(* IEC 61131-3 sources: AXOpen/src/components.rexroth.drives/ctrl/src/AxoCtrlxDriveXsc/v_6_x_x/TypesStructuresAndEnums, 13 files *)

(* ---- AxoCtrlxDriveXsc_Component_Status.st ---- *)
NAMESPACE AXOpen.Components.Rexroth.Drives.v_6_x_x
    {S7.extern=ReadWrite}
    {#ix-attr:[Container(Layout.Stack)]}
    CLASS PUBLIC AxoCtrlxDriveXsc_Component_Status EXTENDS AXOpen.Components.Drives.AxoDrive_Status
        VAR PUBLIC

        END_VAR
    END_CLASS
END_NAMESPACE

(* ---- AxoCtrlxDriveXsc_Config.st ---- *)
NAMESPACE AXOpen.Components.Rexroth.Drives.v_6_x_x
    {S7.extern=ReadWrite}
    {#ix-attr:[Container(Layout.Stack)]}
    CLASS PUBLIC AxoCtrlxDriveXsc_Config
        VAR PUBLIC
            {#ix-set:AttributeName = "<#Info time#>"}
            InfoTime : LTIME := LT#5S;
            {#ix-set:AttributeName = "<#Error time#>"}
            ErrorTime : LTIME := LT#10S;
            {#ix-set:AttributeName = "<#Task timeout#>"}
            TaskTimeout : LTIME := LT#50S;
        END_VAR
    END_CLASS
END_NAMESPACE

(* ---- AxoCtrlxDriveXsc_Control.st ---- *)
NAMESPACE AXOpen.Components.Rexroth.Drives.v_6_x_x
    {S7.extern=ReadWrite}
    {#ix-attr:[Container(Layout.Tabs)]}
    CLASS PUBLIC AxoCtrlxDriveXsc_Control
        VAR PUBLIC
            {#ix-set:AttributeName = "<#DriveControlWord_S_0_0134_0_0#>"}
            DriveControlWord_S_0_0134_0_0 : AxoCtrlxDriveXscDriveControlWord_S_0_0134_0_0;
            {#ix-set:AttributeName = "<#SignalControlWord_S_0_0145_0_0#>"}
            SignalControlWord_S_0_0145_0_0 :    AxoCtrlxDriveXscSignalControlWord_S_0_0145_0_0;
            {#ix-set:AttributeName = "<#CommandPosition_S_0_0282_0_0#>"}
            CommandPosition_S_0_0282_0_0 : DINT;
            {#ix-set:AttributeName = "<#CommandVelocity_S_0_0259_0_0#>"}
            CommandVelocity_S_0_0259_0_0 : DINT;
            {#ix-set:AttributeName = "<#CommandAcceleration_S_0_0260_0_0#>"}
            CommandAcceleration_S_0_0260_0_0 : DINT;
            {#ix-set:AttributeName = "<#CommandDecceleration_S_0_0359_0_0#>"}
            CommandDecceleration_S_0_0359_0_0 : DINT;
            {#ix-set:AttributeName = "<#SupplyUnitControlWord_S_0_1720_0_1#>"}
            SupplyUnitControlWord_S_0_1720_0_1  : AxoCtrlxDriveXscSupplyUnitControlWord_S_0_1720_0_1;
            {#ix-set:AttributeName = "<#BipolarTorqueLimitation_S_0_0092_0_0#>"}
            BipolarTorqueLimitation_S_0_0092_0_0: INT;
            {#ix-set:AttributeName = "<#CommandTorque_S_0_0080_0_0#>"}
            CommandTorque_S_0_0080_0_0 : INT;
            {#ix-set:AttributeName = "<#CommandJerk_S_0_0193_0_0#>"}
            CommandJerk_S_0_0193_0_0 : DINT;
        END_VAR
    END_CLASS
END_NAMESPACE

(* ---- AxoCtrlxDriveXsc_Status.st ---- *)
NAMESPACE AXOpen.Components.Rexroth.Drives.v_6_x_x
    {S7.extern=ReadWrite}
    {#ix-attr:[Container(Layout.Tabs)]}
    CLASS PUBLIC AxoCtrlxDriveXsc_Status
        VAR PUBLIC
            {#ix-set:AttributeName = "<#DriveStatusWord_S_0_0135_0_0#>"}
            DriveStatusWord_S_0_0135_0_0 : AxoCtrlxDriveXscDriveStatusWord_S_0_0135_0_0;
            {#ix-set:AttributeName = "<#SignalStatusWord_S_0_0144_0_0#>"}
            SignalStatusWord_S_0_0144_0_0 : AxoCtrlxDriveXscSignalStatusWord_S_0_0144_0_0;
            {#ix-set:AttributeName = "<#ActualPosition_S_0_0386_0_0#>"}
            ActualPosition_S_0_0386_0_0 : DINT;
            {#ix-set:AttributeName = "<#ActualVelocity_S_0_0535_0_0#>"}
            ActualVelocity_S_0_0535_0_0 : DINT;
            {#ix-set:AttributeName = "<#DiagnosticMessage_S_0_0390_0_0#>"}
            DiagnosticMessage_S_0_0390_0_0 : DWORD;
            {#ix-set:AttributeName = "<#SupplyUnitStatusWord_S_0_1720_0_2#>"}
            SupplyUnitStatusWord_S_0_1720_0_2 : AxoCtrlxDriveXscSupplyUnitStatusWord_S_0_1720_0_2;
            {#ix-set:AttributeName = "<#ActualTorque_S_0_0084_0_0#>"}
            ActualTorque_S_0_0084_0_0 : INT;
        END_VAR
    END_CLASS
END_NAMESPACE

(* ---- AxoCtrlxDriveXscAxisData.st ---- *)
NAMESPACE AXOpen.Components.Rexroth.Drives.v_6_x_x
    {S7.extern=ReadWrite}
    CLASS AxoCtrlxDriveXscAxisData
        VAR PUBLIC
            Cycle                       :   ULINT;
            OverrideVelocityFactor		:	LREAL := 1.0;	//LREAL value to be written
            OverrideAccelerationFactor	:	LREAL := 1.0;	//LREAL value to be written
            OverrideJerkFactor			:	LREAL := 1.0;	//LREAL value to be written
        END_VAR
    END_CLASS
END_NAMESPACE

(* ---- AxoCtrlxDriveXscAxisReference.st ---- *)
// USING AXOpen.Components.Drives;

NAMESPACE AXOpen.Components.Rexroth.Drives.v_6_x_x
    {S7.extern=ReadWrite}
    CLASS AxoCtrlxDriveXscAxisReference IMPLEMENTS AXOpen.Components.Abstractions.Drives.IAxoAxisReference
        VAR PUBLIC // HWin
            {#ix-attr:[Container(Layout.Stack)]}
            {#ix-attr:[ComponentDetails("HW inputs")]}
            {#ix-attr:[ReadOnly()]}
            Inputs  :   AxoCtrlxDriveXsc_Status;
        END_VAR
        VAR PUBLIC // HWout
            {#ix-attr:[Container(Layout.Stack)]}
            {#ix-attr:[ComponentDetails("HW outputs")]}
            // {#ix-attr:[ReadOnly()]}
            Outputs  :   AxoCtrlxDriveXsc_Control;
        END_VAR
        VAR PUBLIC // HWIDs
            {#ix-attr:[Container(Layout.Stack)]}
            {#ix-attr:[ComponentDetails("HWids")]}
            {#ix-attr:[ReadOnly()]}
            HWIDs  :   AxoCtrlxDriveXscHWIDs;
        END_VAR
        VAR PUBLIC // Data
            {#ix-attr:[Container(Layout.Stack)]}
            {#ix-attr:[ComponentDetails("Data")]}
            {#ix-attr:[ReadOnly()]}
            Data            :   AxoCtrlxDriveXscAxisData;
        END_VAR
        VAR PUBLIC
            Config          :   AXOpen.Components.Drives.AxoDrive_Config;
            Status          :   AXOpen.Components.Drives.AxoDrive_Status;
        END_VAR
    END_CLASS
END_NAMESPACE

(* ---- AxoCtrlxDriveXscDriveControlWord_S_0_0134_0_0.st ---- *)
NAMESPACE AXOpen.Components.Rexroth.Drives.v_6_x_x
    {S7.extern=ReadWrite}
    {#ix-attr:[Container(Layout.Wrap)]}
    {#ix-attr:[Group(GroupLayout.GroupBox)]}
    {#ix-set:AttributeName = "<#DriveControlWord#>"}
    CLASS AxoCtrlxDriveXscDriveControlWord_S_0_0134_0_0
        VAR PUBLIC
            {#ix-set:AttributeName = "<#_bit00_Reserve#>"}
            _bit00_Reserve 				:	BOOL;
            {#ix-set:AttributeName = "<#_bit01_Reserve#>"}
            _bit01_Reserve 				:	BOOL;
            {#ix-set:AttributeName = "<#_bit02_Reserve#>"}
            _bit02_Reserve 				:	BOOL;
            {#ix-set:AttributeName = "<#_bit03_Reserve#>"}
            _bit03_Reserve 				:	BOOL;
            {#ix-set:AttributeName = "<#_bit04_Reserve#>"}
            _bit04_Reserve 				:	BOOL;
            {#ix-set:AttributeName = "<#_bit05_Reserve#>"}
            _bit05_Reserve 				:	BOOL;
            {#ix-set:AttributeName = "<#_bit06_Reserve#>"}
            _bit06_Reserve 				:	BOOL;
            {#ix-set:AttributeName = "<#_bit07_Reserve#>"}
            _bit07_Reserve 				:	BOOL;

            {#ix-set:AttributeName = "<#Command operation mode Bit 0#>"}
            CommandOperationModeBit0 	:	BOOL;		//  Command operation mode bit 0                        |   000:  Primary operation mode
                                                        //                                                      |   001:  Secondary operation mode 1
            {#ix-set:AttributeName = "<#Command operation mode Bit 1#>"}
            CommandOperationModeBit1 	:	BOOL;		//  Command operation mode bit 1                        |   010:  Secondary operation mode 2
                                                        //                                                      |   011:  Secondary operation mode 3
                                                        //                                                      |   100:  Secondary operation mode 4
            {#ix-set:AttributeName = "<#Command operation mode Bit 2#>"}
            CommandOperationModeBit2 	:	BOOL;		//  Command operation mode bit 2                        |   101:  Secondary operation mode 5
                                                        //                                                      |   110:  Secondary operation mode 6
                                                        //                                                      |   111:  Secondary operation mode 7
            {#ix-set:AttributeName = "<#_bit11_Reserve#>"}
            _bit11_Reserve 				:	BOOL;
            {#ix-set:AttributeName = "<#_bit12_Reserve#>"}
            _bit12_Reserve 				:	BOOL;
            {#ix-set:AttributeName = "<#Drive Halt#>"}
            DriveHalt 				:	BOOL;		        //  1-0 change: Deceleration of drive while maintaining maximum acceleration (S‑0‑0138 - only possible if bits 14 and 15 = 1)
            {#ix-set:AttributeName = "<#Drive enable#>"}
            DriveEnable 				:	BOOL;		    //  Negative edge: Torque disable without delay (independent of bit 15 or 13)
            {#ix-set:AttributeName = "<#Drive On#>"}
            DriveOn 				:	BOOL;		        //  Negative edge: Best possible deceleration (only possible if bit 14 = 1)
        END_VAR
    END_CLASS
END_NAMESPACE

(* ---- AxoCtrlxDriveXscDriveStatusWord_S_0_0135_0_0.st ---- *)
NAMESPACE AXOpen.Components.Rexroth.Drives.v_6_x_x
    {S7.extern=ReadWrite}
    {#ix-attr:[Container(Layout.Wrap)]}
    {#ix-attr:[Group(GroupLayout.GroupBox)]}
    {#ix-set:AttributeName = "<#DriveStatusWord#>"}
    CLASS AxoCtrlxDriveXscDriveStatusWord_S_0_0135_0_0
        VAR PUBLIC
            {#ix-set:AttributeName = "<#_bit00_Reserve#>"}
            _bit00_Reserve 				:	BOOL;
            {#ix-set:AttributeName = "<#_bit01_Reserve#>"}
            _bit01_Reserve 				:	BOOL;
            {#ix-set:AttributeName = "<#_bit02_Reserve#>"}
            _bit02_Reserve 				:	BOOL;
            {#ix-set:AttributeName = "<#CommandProcessingStatus#>"}
            CommandProcessingStatus		:	BOOL;		//  0 - Drive ignores command value input           |   1 -Drive follows command value input
            {#ix-set:AttributeName = "<#InStandstill#>"}
            InStandstill 				:	BOOL;		//  Drive "Halt" status                             |   1- Act vel < standstill window
            {#ix-set:AttributeName = "<#InReference#>"}
            InReference 				:	BOOL;		//  Drive hommed
            {#ix-set:AttributeName = "<#_bit06_Reserve#>"}
            _bit06_Reserve 				:	BOOL;
            {#ix-set:AttributeName = "<#HardwareLock#>"}
            HardwareLock                :	BOOL;       //  Hardware lock (E-stop)
            {#ix-set:AttributeName = "<#ActualOperatingModeBit0#>"}
            ActualOperatingModeBit0 	:	BOOL;		//  Actual_operating mode bit 0                     |   000:  Primary operation mode
                                                        //                                                  |   001:  Secondary operation mode 1
            {#ix-set:AttributeName = "<#ActualOperatingModeBit1#>"}
            ActualOperatingModeBit1 	:	BOOL;		//  Actual_operating mode bit 1                     |   010:  Secondary operation mode 2
                                                        //                                                  |   011:  Secondary operation mode 3
                                                        //                                                  |   100:  Secondary operation mode 4
            {#ix-set:AttributeName = "<#ActualOperatingModeBit2#>"}
            ActualOperatingModeBit2 	:	BOOL;		//  Actual_operating mode bit 2                     |   101:  Secondary operation mode 5
                                                        //                                                  |   110:  Secondary operation mode 6
                                                        //                                                  |   111:  Secondary operation mode 7
            {#ix-set:AttributeName = "<#_bit11_Reserve#>"}
            _bit11_Reserve 				:	BOOL;
            {#ix-set:AttributeName = "<#WarningZKL2#>"}
            WarningZKL2 				:	BOOL;		//  Warning ZKL2
            {#ix-set:AttributeName = "<#DriveErrorZKL1#>"}
            DriveErrorZKL1 				:	BOOL;		//  Drive Error ZKL1
            {#ix-set:AttributeName = "<#ReadyForOperation Bit 0#>"}
            ReadyForOperationBit0       :	BOOL;		//  Ready to operate bit 0 lower significant bit    |   10: Control section and power section ready for op. (Ab)
                                                        //                                                  |   11: In operation, with torque (e.g. AF)
            {#ix-set:AttributeName = "<#ReadyForOperation Bit 1#>"}
            ReadyForOperationBit1       :	BOOL;		//  Ready to operate bit 1 higher significant bit   |   00: Not ready for power on (e.g., P2)
                                                        //                                                  |   01: Ready for power on (bb)
        END_VAR
    END_CLASS
END_NAMESPACE

(* ---- AxoCtrlxDriveXscHWIDs.st ---- *)
NAMESPACE AXOpen.Components.Rexroth.Drives.v_6_x_x
   {S7.extern=ReadWrite}
	CLASS AxoCtrlxDriveXscHWIDs
      VAR PUBLIC
         {#ix-set:AttributeName = "<#Hardware ID Device#>"}
         HW_Device            : UINT;
         {#ix-set:AttributeName = "<#Hardware ID 'Outputs' module#>"}
         HW_Outputs           : UINT;
         {#ix-set:AttributeName = "<#Hardware ID 'Inputs' module#>"}
         HW_Inputs            : UINT;
         {#ix-set:AttributeName = "<#Hardware ID 'S_0_0134_0_0__Servodrive_profile__Control_word' submodule#>"}
         HW_S_0_0134_0_0      : UINT;
         {#ix-set:AttributeName = "<#Hardware ID 'S_0_0145_0_0__Signal_control_word__Value' submodule#>"}
         HW_S_0_0145_0_0      : UINT;
         {#ix-set:AttributeName = "<#Hardware ID 'S_0_0282_0_0__Drive_controlled_positioning__Command_value' submodule#>"}
         HW_S_0_0282_0_0      : UINT;
         {#ix-set:AttributeName = "<#Hardware ID 'S_0_0259_0_0__Positioning_profile__Profile_velocity' submodule#>"}
         HW_S_0_0259_0_0      : UINT;
         {#ix-set:AttributeName = "<#Hardware ID 'S_0_0260_0_0__Positioning_profile__Acceleration' submodule#>"}
         HW_S_0_0260_0_0      : UINT;
         {#ix-set:AttributeName = "<#Hardware ID 'S_0_0359_0_0__Positioning_profile__Deceleration' submodule#>"}
         HW_S_0_0359_0_0      : UINT;
         {#ix-set:AttributeName = "<#Hardware ID 'S_0_1720_0_1__Power_supply_control__Control_word' submodule#>"}
         HW_S_0_1720_0_1      : UINT;
         {#ix-set:AttributeName = "<#Hardware ID 'S_0_0092_0_0__Torque_force_limitation__Limit_value_bipolar' submodule#>"}
         HW_S_0_0092_0_0      : UINT;
         {#ix-set:AttributeName = "<#Hardware ID 'S_0_0080_0_0__Torque_force_command_value' submodule#>"}
         HW_S_0_0080_0_0      : UINT;
         {#ix-set:AttributeName = "<#Hardware ID 'S_0_0193_0_0__Positioning_jerk' submodule#>"}
         HW_S_0_0193_0_0      : UINT;
         {#ix-set:AttributeName = "<#Hardware ID 'S_0_0135_0_0__Servodrive_profile__Status_word' submodule#>"}
         HW_S_0_0135_0_0      : UINT;
         {#ix-set:AttributeName = "<#Hardware ID 'S_0_0144_0_0__Signal_status_word__Value' submodule#>"}
         HW_S_0_0144_0_0      : UINT;
         {#ix-set:AttributeName = "<#Hardware ID 'S_0_0386_0_0__Position_controller__Position_actual_value' submodule#>"}
         HW_S_0_0386_0_0      : UINT;
         {#ix-set:AttributeName = "<#Hardware ID 'S_0_0535_0_0__Velocity_controller__Velocity_actual_value' submodule#>"}
         HW_S_0_0535_0_0      : UINT;
         {#ix-set:AttributeName = "<#Hardware ID 'S_0_0390_0_0__Diagnostic_message__Manufacturer_status_register' submodule#>"}
         HW_S_0_0390_0_0      : UINT;
         {#ix-set:AttributeName = "<#Hardware ID 'S_0_1720_0_2__Power_supply_control__Status_word' submodule#>"}
         HW_S_0_1720_0_2      : UINT;
         {#ix-set:AttributeName = "<#Hardware ID 'S_0_0084_0_0__Torque_force_feedback_value' submodule#>"}
         HW_S_0_0084_0_0      : UINT;
         {#ix-set:AttributeName = "<#Hardware ID 'P_0_0106_0_0__STO_function__Operating_status' submodule#>"}
         HW_P_0_0106_0_0      : UINT;
      END_VAR
   END_CLASS
END_NAMESPACE

(* ---- AxoCtrlxDriveXscSignalControlWord_S_0_0145_0_0.st ---- *)
NAMESPACE AXOpen.Components.Rexroth.Drives.v_6_x_x
    {S7.extern=ReadWrite}
    {#ix-attr:[Container(Layout.Wrap)]}
    {#ix-attr:[Group(GroupLayout.GroupBox)]}
    {#ix-set:AttributeName = "<#SignalControlWord#>"}
    CLASS AxoCtrlxDriveXscSignalControlWord_S_0_0145_0_0
        VAR PUBLIC
            {#ix-set:AttributeName = "<#Acceptance of positioning command value#>"}
            AcceptanceOfPositioningCommandValue:	BOOL;		                                    //  Bit 0 of the Drive-controlled positioning: Control word (S-0-0346) !!! must be set in drive !!!
            {#ix-set:AttributeName = "<#_bit01_Reserve#>"}
            _bit01_Reserve 				:	BOOL;
            {#ix-set:AttributeName = "<#Homing control#>"}
            HomingControl 				:	BOOL;		                                            //  Bit 0 of the Homing control: C0600 Command drive-controlled procedure (S-0-0148) !!! must be set in drive !!!
            {#ix-set:AttributeName = "<#Absolute/Relative type of positioning command value#>"}
            AbsoluteRelative 				:	BOOL;				                                //  Bit 3 of the Drive-controlled positioning: Control word (S-0-0346) !!! must be set in drive !!!
            {#ix-set:AttributeName = "<#Immediate block change#>"}
            ImmediateChange 				:	BOOL;                                               //  Bit 5 of the Drive-controlled positioning: Control word (S-0-0346) !!! must be set in drive !!!
            {#ix-set:AttributeName = "<#Clear error#>"}
            ClearError  :	BOOL;                                                                   //  Bit 0 of the Class 1 diagnostics: C0500 Reset command (S-0-0099) !!! must be set in drive !!!
            {#ix-set:AttributeName = "<#Infinite travel in positive direction (jog+)#>"}
            JogPositive :	BOOL;                                                                   //  Bit 1 of the Drive-controlled positioning: Control word (S-0-0346) !!! must be set in drive !!!
            {#ix-set:AttributeName = "<#Infinite travel in negative direction (jog-)#>"}
            JogNegative :	BOOL;                                                                   //  Bit 2 of the Drive-controlled positioning: Control word (S-0-0346) !!! must be set in drive !!!
            {#ix-set:AttributeName = "<#Activate configuration mode#>"}
            SwitchToCM  :	BOOL;                                                                   //  Bit 0 of the Subdevice STM: C0400 Activate configuration mode (S-0-0420) !!! must be set in drive !!!
            {#ix-set:AttributeName = "<#Activate operation mode#>"}
            SwitchTo0M  :	BOOL;                                                                   //  Bit 0 of the Subdevice STM: C0200 Activate operation mode (S-0-0422) !!! must be set in drive !!!
            {#ix-set:AttributeName = "<#CancelReferencePoint#>"}
            CancelReferencePoint        :	BOOL;		                                            // Homing function: C1500 Command cancel reference point (0x2500:01 / S-0-0191 / --) !!! must be set in drive !!!
            {#ix-set:AttributeName = "<#Device reboot#>"}
            DeviceReboot 				:	BOOL;
            {#ix-set:AttributeName = "<#_bit12_Reserve#>"}
            _bit12_Reserve 				:	BOOL;
            {#ix-set:AttributeName = "<#_bit13_Reserve#>"}
            _bit13_Reserve 				:	BOOL;
            {#ix-set:AttributeName = "<#_bit14_Reserve#>"}
            _bit14_Reserve 				:	BOOL;
            {#ix-set:AttributeName = "<#Set absolute position function#>"}
            SetAbsPositionFunction  :	BOOL;                                                       //  Bit 0 of the Set absolute position function: C0300 Command procedure (S-0-0447) !!! must be set in drive !!!
        END_VAR
    END_CLASS
END_NAMESPACE

(* ---- AxoCtrlxDriveXscSignalStatusWord_S_0_0144_0_0.st ---- *)
NAMESPACE AXOpen.Components.Rexroth.Drives.v_6_x_x
    {S7.extern=ReadWrite}
    {#ix-attr:[Container(Layout.Wrap)]}
    {#ix-attr:[Group(GroupLayout.GroupBox)]}
    {#ix-set:AttributeName = "<#SignalStatusWord#>"}
    CLASS AxoCtrlxDriveXscSignalStatusWord_S_0_0144_0_0
        VAR PUBLIC
            {#ix-set:AttributeName = "<#Configuration/Parametrization/Operation bit 0#>"}
            CmPmOmBit0 				:	BOOL;		//  Bit 0 of the Subdevice STM: Status, parameterization mode (S-0-0424)  !!! must be set in drive !!!
            {#ix-set:AttributeName = "<#Configuration/Parametrization/Operation bit 1#>"}
            CmPmOmBit1 				:	BOOL;		//  Bit 1 of the Subdevice STM: Status, parameterization mode (S-0-0424)  !!! must be set in drive !!!
            {#ix-set:AttributeName = "<#In target position#>"}
            InTargetPosition 				:	BOOL;		//  Bit 2 of the Positioning status: Word (S-0-0437)  !!! must be set in drive !!!
            {#ix-set:AttributeName = "<#Position command acknowledgment#>"}
            PositionCommandAck 				:	BOOL;		//  Bit 0 of the Drive-controlled positioning: Command acknowledgment (S-0-0419)  !!! must be set in drive !!!
            {#ix-set:AttributeName = "<#Drive standstill#>"}
            DriveStandstill 				:	BOOL;		//  Bit 0 of the Velocity status: Actual value = 0 (S-0-0331)  !!! must be set in drive !!!
            {#ix-set:AttributeName = "<#Command change bit#>"}
            CommandChangeBit 				:	BOOL;		//  Bit 5 of the Axis state machine: Status word, axis (P-0-0115 )  !!! must be set in drive !!!
            {#ix-set:AttributeName = "<#_bit6_Reserve#>"}
            _bit6_Reserve 				:	BOOL;
            {#ix-set:AttributeName = "<#_bit7_Reserve#>"}
            _bit7_Reserve 				:	BOOL;
            {#ix-set:AttributeName = "<#Locked by hardware#>"}
            LockedByHardware            :	BOOL;		    //  Bit 7 of the Axis state machine: Status word 2, axis (P-0-0110 )  !!! must be set in drive !!!
            {#ix-set:AttributeName = "<#_bit9_Reserve#>"}
            _bit9_Reserve 				:	BOOL;
            {#ix-set:AttributeName = "<#_bit10_Reserve#>"}
            _bit10_Reserve 				:	BOOL;
            {#ix-set:AttributeName = "<#_bit11_Reserve#>"}
            _bit11_Reserve 				:	BOOL;
            {#ix-set:AttributeName = "<#_bit12_Reserve#>"}
            _bit12_Reserve 				:	BOOL;
            {#ix-set:AttributeName = "<#_bit13_Reserve#>"}
            _bit13_Reserve 				:	BOOL;
            {#ix-set:AttributeName = "<#_bit14_Reserve#>"}
            _bit14_Reserve 				:	BOOL;
            {#ix-set:AttributeName = "<#_bit15_Reserve#>"}
            _bit15_Reserve 				:	BOOL;
        END_VAR
    END_CLASS
END_NAMESPACE

(* ---- AxoCtrlxDriveXscSupplyUnitControlWord_S_0_1720_0_1.st ---- *)
NAMESPACE AXOpen.Components.Rexroth.Drives.v_6_x_x
    {S7.extern=ReadWrite}
    {#ix-attr:[Container(Layout.Wrap)]}
    {#ix-attr:[Group(GroupLayout.GroupBox)]}
    {#ix-set:AttributeName = "<#SupplyUnitControlWord#>"}
    CLASS AxoCtrlxDriveXscSupplyUnitControlWord_S_0_1720_0_1
        VAR PUBLIC
            {#ix-set:AttributeName = "<#_bit0_Reserve#>"}
            _bit0_Reserve 				:	BOOL;
            {#ix-set:AttributeName = "<#_bit1_Reserve#>"}
            _bit1_Reserve 				:	BOOL;
            {#ix-set:AttributeName = "<#_bit2_Reserve#>"}
            _bit2_Reserve 				:	BOOL;
            {#ix-set:AttributeName = "<#_bit3_Reserve#>"}
            _bit3_Reserve 				:	BOOL;
            {#ix-set:AttributeName = "<#_bit4_Reserve#>"}
            _bit4_Reserve 				:	BOOL;
            {#ix-set:AttributeName = "<#_bit4_Reserve#>"}
            _bit5_Reserve 				:	BOOL;
            {#ix-set:AttributeName = "<#_bit6_Reserve#>"}
            _bit6_Reserve 				:	BOOL;
            {#ix-set:AttributeName = "<#_bit7_Reserve#>"}
            _bit7_Reserve 				:	BOOL;
            {#ix-set:AttributeName = "<#Mode selection bit 0#>"}
            ModeSelectionBit0 	:	BOOL;		                    //  Mode selection bit 0                                |   00:  Primary operation mode
                                                                    //                                                      |   01:  1 secondary operation mode
            {#ix-set:AttributeName = "<#Mode selection bit 1#>"}
            ModeSelectionBit1 	:	BOOL;		                    //  Command operation mode bit 1                        |   10:  2 secondary operation mode
                                                                    //                                                      |   11:  3 secondary operation mode
            {#ix-set:AttributeName = "<#DC bus discharge#>"}
            DCbusDischarge  :   BOOL;                               //  0: DC bus discharge not active
                                                                    //  1: Start DC bus discharge function
            {#ix-set:AttributeName = "<#_bit11_Reserve#>"}
            _bit11_Reserve 				:	BOOL;
            {#ix-set:AttributeName = "<#Controlling the ready for operation relay#>"}
            ControllingTheReadyForOperationRelay    :	BOOL;       //  0: Open contact
                                                                    //  1: Close contact, release
            {#ix-set:AttributeName = "<#_bit13_Reserve#>"}
            _bit13_Reserve 				:	BOOL;
            {#ix-set:AttributeName = "<#Controlling DC bus charging and mains contactor#>"}
            ControllingDCbusChargingAndMainsContactor   :	BOOL;   //  0: Mains disconnection e.g. by opening the mains contactor or by locking the mains thyristors
                                                                    //  1: Charge DC bus by closing the mains contactor or by activating the mains thyristors - device goes into rectifier mode
            {#ix-set:AttributeName = "<#Enabling#>"}
            Enabling:	BOOL;                                       //  0: Disabled, command operation mode not active
                                                                    //  1: Enabled, command operation mode active
        END_VAR
    END_CLASS
END_NAMESPACE

(* ---- AxoCtrlxDriveXscSupplyUnitStatusWord_S_0_1720_0_2.st ---- *)
NAMESPACE AXOpen.Components.Rexroth.Drives.v_6_x_x
    {S7.extern=ReadWrite}
    {#ix-attr:[Container(Layout.Wrap)]}
    {#ix-attr:[Group(GroupLayout.GroupBox)]}
    {#ix-set:AttributeName = "<#SupplyUnitStatusWord#>"}
    CLASS AxoCtrlxDriveXscSupplyUnitStatusWord_S_0_1720_0_2
        VAR PUBLIC
            {#ix-set:AttributeName = "<#_bit0_Reserve#>"}
            _bit0_Reserve 				:	BOOL;
            {#ix-set:AttributeName = "<#_bit1_Reserve#>"}
            _bit1_Reserve 				:	BOOL;
            {#ix-set:AttributeName = "<#_bit2_Reserve#>"}
            _bit2_Reserve 				:	BOOL;
            {#ix-set:AttributeName = "<#_bit3_Reserve#>"}
            _bit3_Reserve 				:	BOOL;
            {#ix-set:AttributeName = "<#Mains status#>"}
            MainsStatus				:	BOOL;
            {#ix-set:AttributeName = "<#Hardware enable#>"}
            HardwareEnable				:	BOOL;
            {#ix-set:AttributeName = "<#Controlling the mains connection#>"}
            ControllingTheMainsConnection				:	BOOL;
            {#ix-set:AttributeName = "<#Bb contact#>"}
            BbContact				:	BOOL;
            {#ix-set:AttributeName = "<#Feedback of the preselected operation modes bit 0#>"}   //  00: Primary operation mode
            PreselectedOPmodesFB_bit0    :	BOOL;                                               //  10: Secondary operation mode 2
            {#ix-set:AttributeName = "<#Feedback of the preselected operation modes bit 1#>"}   //  11: Secondary operation mode 3
            PreselectedOPmodesFB_bit01      :	BOOL;
            {#ix-set:AttributeName = "<#DC bus discharge#>"}
            DCbusDischarge  :	BOOL;
            {#ix-set:AttributeName = "<#Braking resistor#>"}
            BrakingResistor  :	BOOL;
            {#ix-set:AttributeName = "<#Warning#>"}
            Warning  :	BOOL;
            {#ix-set:AttributeName = "<#Error#>"}
            Error  :	BOOL;
            {#ix-set:AttributeName = "<#Ready for enabling#>"}
            ReadyForEnabling:	BOOL;
            {#ix-set:AttributeName = "<#Enabling#>"}
            Enabling:	BOOL;
        END_VAR
    END_CLASS
END_NAMESPACE
